// TwinCAT 3 PLC project PLC
// ProgramVersion: 3.1.4024.0
// libraries:
//   Tc2_Standard, * (Beckhoff Automation GmbH)
//   Tc2_System, * (Beckhoff Automation GmbH)
//   Tc3_Module, * (Beckhoff Automation GmbH)
// project tree:
//   DUTs/ ST_Point.TcDUT
//   GVLs/ GVL.TcGVL
//   / PlcTask.TcTTO
//   POUs/ MAIN.TcPOU
// real-time tasks:
//   TASK PlcTask: cycle T#10ms, priority 20, ADS port 350

CONFIGURATION PLC
    RESOURCE PLC ON TwinCAT3
        TASK PlcTask(INTERVAL := T#10ms, PRIORITY := 20);
        PROGRAM MAIN WITH PlcTask : MAIN;
    END_RESOURCE
END_CONFIGURATION

// ---- DUTs/ST_Point.TcDUT
TYPE ST_Point :
STRUCT
	x		: LREAL;
	y		: LREAL;
END_STRUCT
END_TYPE

// ---- GVLs/GVL.TcGVL
{attribute 'qualified_only'}
VAR_GLOBAL
	Points		: ARRAY[0..9] OF ST_Point;
END_VAR

// ---- POUs/MAIN.TcPOU
PROGRAM MAIN
VAR
	Position		: LREAL;
	Velocity		: LREAL;
	
	rand			: ARRAY[0..1] OF DRAND;
	i				: INT;
	ton				: TON;
	
	iWriteMe		: DINT := 0;
END_VAR

ton(IN:=NOT ton.Q, PT:=T#1S);
IF ton.Q THEN
	FOR i := 0 TO 1 DO
		rand[i](Seed:=i);
	END_FOR
	
	Position := Position + rand[0].Num;
	Velocity := rand[1].Num * 100;
END_IF

END_PROGRAM
